{attribute 'qualified_only'}
VAR_GLOBAL
END_VAR

(* stored: Version 1.1.0.1, ProductVersion 3.1.4024.4
   GVL Outputs: Id {5acb3c89-0324-4f89-9479-b7ab57d55ca9} *)
